(* IEC 61131-3 sources: codesys-mcp-toolkit/standalone-sync/sources_st/511_05/FUNCs, 3 files *)

(* ---- F_ElemerREM_Flow.func.st ---- *)
// @OBJECT_ID: 22b7d66b-5897-4426-b661-360de4c0c760
// @DECLARATION
(* Мгновенный расход F2: 2 регистра WORD, Big-Endian REAL *)
FUNCTION F_ElemerREM_Flow : REAL
VAR_INPUT
    pBuf : POINTER TO ARRAY[0..1] OF WORD;
END_VAR
VAR
    dw : DWORD;
	END_VAR

// @IMPLEMENTATION
IF pBuf <> 0 THEN
    // Склеиваем два WORD в один DWORD (старшее слово сдвигаем на 16 бит влево)
    dw := SHL(WORD_TO_DWORD(pBuf^[0]), 16) OR WORD_TO_DWORD(pBuf^[1]);

    // Копируем память "бит-в-бит" из DWORD в REAL
    SysMemCpy(pDest := ADR(F_ElemerREM_Flow), pSrc := ADR(dw), udiCount := 4);
END_IF

(* ---- F_ElemerREM_Volume.func.st ---- *)
// @OBJECT_ID: 4d85027d-cb35-4b94-8eef-0ae63feaf4df
// @DECLARATION
(*  Накопленный объём F1: 4 регистра WORD, Big-Endian Double → REAL  *)
FUNCTION F_ElemerREM_Volume : REAL
VAR_INPUT
    pBuf : POINTER TO ARRAY[0..3] OF WORD;
END_VAR
VAR
    lr   : LREAL;
    pW   : POINTER TO WORD;
END_VAR

// @IMPLEMENTATION
pW    := ADR(lr);
pW[3] := pBuf^[0];
pW[2] := pBuf^[1];
pW[1] := pBuf^[2];
pW[0] := pBuf^[3];
F_ElemerREM_Volume := LREAL_TO_REAL(lr);

(* ---- F_GetReal_BADC.func.st ---- *)
// @OBJECT_ID: b25eaad9-59ce-4c23-9aa6-5c998f777003
// @DECLARATION
(*
    ФУНКЦИЯ: F_GetReal_BADC
    ОПИСАНИЕ: Разбор REAL 32 бита из 2 регистров WORD, порядок байт BADC.

    Прибор передаёт байты в порядке: B A D C
    (где ABCD = нормальный Big-Endian порядок)

    Раскладка по байтам:
      pSrc[0] = B,  pSrc[1] = A,  pSrc[2] = D,  pSrc[3] = C

    Для Little-Endian ЦПУ нужно собрать DCBA:
      pDst[0] = C = pSrc[3]
      pDst[1] = D = pSrc[2]
      pDst[2] = A = pSrc[1]
      pDst[3] = B = pSrc[0]
*)
FUNCTION F_GetReal_BADC : REAL
VAR_INPUT
    pBuf : POINTER TO ARRAY[0..1] OF WORD;
END_VAR
VAR
    dw   : DWORD;
    pSrc : POINTER TO BYTE;
    pDst : POINTER TO BYTE;
END_VAR

// @IMPLEMENTATION

pSrc    := ADR(pBuf^[0]);
pDst    := ADR(dw);
pDst[0] := pSrc[3]; // C
pDst[1] := pSrc[2]; // D
pDst[2] := pSrc[1]; // A
pDst[3] := pSrc[0]; // B
SysMemCpy(pDest := ADR(F_GetReal_BADC), pSrc := ADR(dw), udiCount := 4);
